# EPICS substitutions: iocs/testM4/testM4App/Db/testM4_expanded.substitutions
# This file was automatically generated on Thu 26 May 2016 16:08:02 BST from
# source: /home/hgv27681/R3.14.12.3/support/smaractEcm/etc/makeIocs/testM4.xml
#
# *** Please do not edit this file: edit the source file instead. ***
#

# Macros:
#  P        EPICS name prefix
#  R        EPICS name suffix
#  PORT     Asyn port
#  TIMEOUT  Timeout
file $(SMARACTECM)/db/smaractEcmController.template
{
pattern { P, R, PORT, TIMEOUT }
    { "BL21I-MO-POD-01", ":ECM1", "ecm1", "0" }
}

file $(SMARACTECM)/db/smarpodAxis.template
{
pattern { P, R, PORT, AXIS, TIMEOUT }
    { "BL21I-MO-POD-01:A", "X", "ecm1", "0", "1" }
    { "BL21I-MO-POD-01:A", "Y", "ecm1", "1", "1" }
    { "BL21I-MO-POD-01:A", "Z", "ecm1", "2", "1" }
    { "BL21I-MO-POD-01:A", "RX", "ecm1", "3", "1" }
    { "BL21I-MO-POD-01:A", "RY", "ecm1", "4", "1" }
    { "BL21I-MO-POD-01:A", "RZ", "ecm1", "5", "1" }
}

# Macros:
#  P           Device Prefix
#  M           Device Suffix
#  PORT        Asyn port for motor record
#  ADDR        Address on controller
#  DESC        Description, displayed on EDM screen
#  MRES        Motor Step Size (EGU)
#  VELO        Velocity (EGU/s)
#  PREC        Display Precision
#  EGU         Engineering Units
#  TWV         Tweak Step Size (EGU)
#  DTYP        DTYP of record
#  DIR         User Direction
#  VBAS        Base Velocity (EGU/s)
#  VMAX        Max Velocity (EGU/s), defaults to VELO
#  ACCL        Seconds to Velocity
#  BDST        BL Distance (EGU)
#  BVEL        BL Velocity (EGU/s)
#  BACC        BL Seconds to Veloc.
#  DHLM        Dial High Limit
#  DLLM        Dial Low Limit
#  HLM         User High Limit
#  LLM         User Low Limit
#  HLSV        HW Lim. Violation Svr
#  INIT        Startup commands
#  SREV        Steps per Revolution
#  RRES        Readback Step Size (EGU)
#  ERES        Encoder Step Size (EGU)
#  JAR         Jog Acceleration (EGU/s^2)
#  UEIP        Use Encoder If Present
#  URIP        Use RDBL If Present
#  RDBL        Readback Location, set URIP = 1 if you specify this
#  RTRY        Max retry count
#  DLY         Readback settle time (s)
#  OFF         User Offset (EGU)
#  RDBD        Retry Deadband (EGU)
#  FOFF        Freeze Offset, 0=variable, 1=frozen
#  ADEL        Alarm monitor deadband (EGU)
#  NTM         New Target Monitor, only set to 0 for soft motors
#  FEHIGH      HIGH limit for following error
#  FEHIHI      HIHI limit for following error
#  FEHHSV      HIHI alarm severity for following error
#  FEHSV       HIGH alarm severity for following error
#  SCALE       Scale factor, if pmacSetAxisScale is used this should be set
#  HOMEVIS     If 1 then home is visible on the gui
#  HOMEVISSTR  If HOMEVIS=0, then display this text on the gui instead
#  name        Object name and gui association name
#  alh         Set this to alh to add the motor to the alarm handler and send emails,
#  gda_name    Name to export this as to GDA
#  gda_desc    Description to export this as to GDA
file $(MOTOR)/db/basic_asyn_motor.template
{
pattern { P, M, PORT, ADDR, DESC, MRES, VELO, PREC, EGU, TWV, DTYP, DIR, VBAS, VMAX, ACCL, BDST, BVEL, BACC, DHLM, DLLM, HLM, LLM, HLSV, INIT, SREV, RRES, ERES, JAR, UEIP, URIP, RDBL, RTRY, DLY, OFF, RDBD, FOFF, ADEL, NTM, FEHIGH, FEHIHI, FEHHSV, FEHSV, SCALE, HOMEVIS, HOMEVISSTR, name, alh, gda_name, gda_desc }
    { "BL21I-MO-POD-01", ":X", "ecm1", "0", "X Translation", ".001", "50", "5", "um", "10", "asynMotor", "0", "0", "$(VELO)", "0.5", "0", "0", "", "80000000", "-80000000", "", "", "MAJOR", "", "200", "", "", "", "0", "0", "", "0", "0", "0", "", "0", "0", "1", "0", "0", "NO_ALARM", "NO_ALARM", "1", "1", "Use motor summary screen", "S1X", "None", "X", "$(DESC)" }
    { "BL21I-MO-POD-01", ":Y", "ecm1", "1", "Y Translation", ".001", "50", "5", "um", "10", "asynMotor", "0", "0", "$(VELO)", "0.5", "0", "0", "", "80000000", "-80000000", "", "", "MAJOR", "", "200", "", "", "", "0", "0", "", "0", "0", "0", "", "0", "0", "1", "0", "0", "NO_ALARM", "NO_ALARM", "1", "1", "Use motor summary screen", "S1Y", "None", "Y", "$(DESC)" }
    { "BL21I-MO-POD-01", ":Z", "ecm1", "2", "Z Translation", ".001", "50", "5", "um", "10", "asynMotor", "0", "0", "$(VELO)", "0.5", "0", "0", "", "80000000", "-80000000", "", "", "MAJOR", "", "200", "", "", "", "0", "0", "", "0", "0", "0", "", "0", "0", "1", "0", "0", "NO_ALARM", "NO_ALARM", "1", "1", "Use motor summary screen", "S1Z", "None", "Z", "$(DESC)" }
    { "BL21I-MO-POD-01", ":RX", "ecm1", "3", "X Rotation", ".001", "50", "5", "udeg", "10", "asynMotor", "0", "0", "$(VELO)", "0.5", "0", "0", "", "80000000", "-80000000", "", "", "MAJOR", "", "200", "", "", "", "0", "0", "", "0", "0", "0", "", "0", "0", "1", "0", "0", "NO_ALARM", "NO_ALARM", "1", "1", "Use motor summary screen", "S1RX", "None", "RX", "$(DESC)" }
    { "BL21I-MO-POD-01", ":RY", "ecm1", "4", "Y Rotation", ".001", "50", "5", "udeg", "10", "asynMotor", "0", "0", "$(VELO)", "0.5", "0", "0", "", "80000000", "-80000000", "", "", "MAJOR", "", "200", "", "", "", "0", "0", "", "0", "0", "0", "", "0", "0", "1", "0", "0", "NO_ALARM", "NO_ALARM", "1", "1", "Use motor summary screen", "S1RY", "None", "RY", "$(DESC)" }
    { "BL21I-MO-POD-01", ":RZ", "ecm1", "5", "Z Rotation", ".001", "50", "5", "udeg", "10", "asynMotor", "0", "0", "$(VELO)", "0.5", "0", "0", "", "80000000", "-80000000", "", "", "MAJOR", "", "200", "", "", "", "0", "0", "", "0", "0", "0", "", "0", "0", "1", "0", "0", "NO_ALARM", "NO_ALARM", "1", "1", "Use motor summary screen", "S1RZ", "None", "RZ", "$(DESC)" }
}
